TYPE U_MbConv :
UNION
	lw : LWORD;
	dw : DWORD;
	w  : WORD;
	i  : INT;
	di : DINT;
	li : LINT;
	fR : REAL;
	fL : LREAL;
END_UNION
END_TYPE

(* stored: Version 1.1.0.1
   DUT U_MbConv: Id {b1ffb4e0-d85c-4ed9-9eaa-1f72596c1e2a} *)
